// TIA Portal V16 export
// export: Created 2025-12-30T17:36:41.7055085Z, ExportSetting WithDefaults, DisplayName Totally Integrated Automation Portal, DisplayVersion V16, DisplayName TIA Portal Version Control Interface, DisplayVersion V16, DisplayName TIA Portal Openness, DisplayVersion V16, DisplayName STEP 7 Professional, DisplayVersion V16, DisplayName STEP 7 Safety, DisplayVersion V16, DisplayName WinCC Professional, DisplayVersion V16
VAR_GLOBAL   // PLC tag table "Tag table from XML_1"
   "Moving X" AT %I0.0 : Bool;
   "Moving Z" AT %I0.1 : Bool;
   "Item detected" AT %I0.2 : Bool;
   "Lid at place" AT %I0.3 : Bool;
   "Lid clamped" AT %I0.4 : Bool;
   "Pos. at limit (lids)" AT %I0.5 : Bool;
   "Base at place" AT %I0.6 : Bool;
   "Base clamped" AT %I0.7 : Bool;
   "Pos. at limit (bases)" AT %I1.0 : Bool;
   "Part leaving" AT %I1.1 : Bool;
   Start AT %I1.2 : Bool;
   Reset AT %I1.3 : Bool;
   Stop AT %I1.4 : Bool;
   "Emergency stop" AT %I1.5 : Bool;
   Auto AT %I1.6 : Bool;
   "FACTORY I/O (Uruchomiony)" AT %I1.7 : Bool;
   "Move X" AT %Q0.0 : Bool;
   "Move Z" AT %Q0.1 : Bool;
   Grab AT %Q0.2 : Bool;
   "Lids conveyor" AT %Q0.3 : Bool;
   "Clamp lid" AT %Q0.4 : Bool;
   "Pos. raise (lids)" AT %Q0.5 : Bool;
   "Bases conveyor" AT %Q0.6 : Bool;
   "Clamp base" AT %Q0.7 : Bool;
   "Pos. raise (bases)" AT %Q1.0 : Bool;
   "Start light" AT %Q1.1 : Bool;
   "Reset light" AT %Q1.2 : Bool;
   "Stop light" AT %Q1.3 : Bool;
   "Counter" AT %QD30 : DInt;
END_VAR
